{attribute 'enable_dynamic_creation'}
TYPE Node :
STRUCT
	data : INT;
	pNext : POINTER TO INT;
	pPrev : POINTER TO INT;
END_STRUCT
END_TYPE

(* stored: Version 1.1.0.1
   DUT Node: Id {69e86ae3-d4a3-4140-87f7-f6d7bc87dba3} *)
